{attribute addProperty BoxType "AT2040-0250-0022"}
{attribute addProperty Id "A_0107_AT2000_5233_0018_AT2000_5233AT2000_C5E5984862678.25"}
{attribute addProperty CRC "2535270189"}
{attribute addProperty SizeInBites "626"}
{attribute addProperty SizeInBytes "78.25"}
TYPE A_0037_AT2040_0250_0022_971D272D EXTENDS AT2040_BA5A9548 :
STRUCT
	{attribute addProperty Name "A_0107_AT2000_5233_0018_AT2000_5233"}
	A_0107_AT2000_5233_0018_AT2000_5233 : AT2000_C5E59848;
END_STRUCT
END_TYPE

(* stored: Version 1.2.0.0, ProductVersion 3.1.4024.9
   DUT A_0037_AT2040_0250_0022_971D272D: Id {52eedad6-04ea-4d89-9fca-b90ed04e75fb} *)
